// TIA Portal V17 export
// export: Created 2022-07-20T07:01:26.0319135Z, ExportSetting WithDefaults, DisplayName Totally Integrated Automation Portal, DisplayVersion V17, DisplayName TIA Portal Openness, DisplayVersion V17, DisplayName TIA Portal Version Control Interface, DisplayVersion V17, DisplayName SINAMICS Startdrive Advanced, DisplayVersion V17, DisplayName SINAMICS Startdrive G130, G150, S120, S150, SINAMICS MV, S210, DisplayVersion V17, DisplayName SINAMICS Startdrive G110M, G120, G120C, G120D, G120P, G115D, DisplayVersion V17, DisplayName STEP 7 Professional, DisplayVersion V17, DisplayName STEP 7 Safety, DisplayVersion V17, DisplayName WinCC Advanced, DisplayVersion V17
FUNCTION_BLOCK "FB10233_LAM_PositionningMotor"   // FB10233, LAD
{ S7_Optimized_Access := 'TRUE' }
VERSION : 0.1
// stored: AutoNumber false, IsIECCheckEnabled false, IsRetainMemResEnabled false, MemoryReserve 100, SetENOAutomatically false, UDAEnableTagReadback false
   VAR_INPUT
      DriveInLexium : "TLexium_MDrv_Drv2Plc";
      HomingSensor : Bool;
      MmByMotorTurn : LReal;
      HoldCurrent : SInt;
      RunCurrent : SInt;
      HomingSpeedMmBySec : Real;
      SpeedMmBySec : Real;
      AccelerationMmBySec2 : Real;
      DecelerationMmBySec2 : Real;
      JogSpeedMmBySec : Real;
      OriginPosition : Real;
      StandByPosition : Real;
      WorkingPosition : Real;
   END_VAR
   VAR_OUTPUT
      ActualPosition : Real;
      HomingInProgress : Bool;
      HomingDone : Bool;
      InOriginPosition : Bool;
      IsInStandByPosition : Bool;
      InWorkingPosition : Bool;
      MotorInError : Bool;
      ErrorCode : Array[0..9] of UInt;
   END_VAR
   VAR_IN_OUT
      DriveOutLexium : "TLexium_MDrv_Plc2Drv";
      RequestAcknowledge : Bool;
      RequestHoming : Bool;
      RequestGoToOriginPosition : Bool;
      RequestGoToStandByPosition : Bool;
      RequestGoToWorkingPosition : Bool;
      RequestStop : Bool;
   END_VAR
   VAR
      Motor_Struct : Struct
         In : Struct
            EnableMotor : Bool;
            MmByTurn : LReal;
            "HomingVelocity_mm.s-1" : Real;
            "Velocity_mm.s-1" : Real;
            "Acceleration_mm.s-2" : Real;
            "Deceleration_mm.s-2" : Real;
            "JogVelocity_mm.s-1" : Real;
            RequestHoming : Bool;
            RequestGoToPosition_1 : Bool;
            Position_1 : Real;
            RequestGoToPosition_2 : Bool;
            Position_2 : Real;
            RequestGoToPosition_3 : Bool;
            Position_3 : Real;
            RequestGoToPosition_4 : Bool;
            Position_4 : Real;
            RequestGoToPosition_5 : Bool;
            Position_5 : Real;
            RequestJogPositive : Bool;
            RequestJogNegative : Bool;
            Ack : Bool;
            RequestStop : Bool;
         END_STRUCT;
         Out : Struct
            ActualPosition_mm : Real;
            MotorEnabled : Bool;
            HomingInProgress : Bool;
            HomingDone : Bool;
            IsInPosition_1 : Bool;
            IsInPosition_2 : Bool;
            IsInPosition_3 : Bool;
            IsInPosition_4 : Bool;
            IsInPosition_5 : Bool;
            InError : Bool;
            ErrorCode : Array[0..9] of UInt;
         END_STRUCT;
      END_STRUCT;
      SendRequestAfterEnableOk : Bool;
      SendNewRequestOk : Bool;
      MotorMovementManagementStateDiagram : Int;
      R_TRIG_HomingSensor : R_TRIG;
      R_TRIG_RequestHoming : R_TRIG;
      R_TRIG_RequestGoToOriginPosition : R_TRIG;
      R_TRIG_RequestGoToRecoveryPosition { S7_SetPoint := 'True'} : R_TRIG;
      R_TRIG_RequestGoToWorkingPosition : R_TRIG;
      R_TRIG_HomingDone { S7_SetPoint := 'True'} : R_TRIG;
      TON_Motor_SendRequestAfterEnabled { S7_SetPoint := 'True'} : TON_TIME;
      TON_Motor_SendNewRequest { S7_SetPoint := 'True'} : TON_TIME;
      FB10234_LexiumMotor_Instance { S7_SetPoint := 'True'} : "FB10234_LexiumMotor";
   END_VAR
   VAR CONSTANT
      WAIT_FOR_MOTOR_MOVEMENT_REQUESTS : Int := 0;
      MOTOR_HOMING : Int := 10;
      MOTOR_GO_TO_ORIGIN_POSITION : Int := 20;
      MOTOR_GO_TO_RECOVERY_POSITION : Int := 30;
      MOTOR_GO_TO_WORKING_POSITION : Int := 40;
      MOTOR_MOVEMENT_REQUEST_DONE : Int := 50;
   END_VAR
BEGIN

REGION Network 1 (SCL): First Scan
   IF "FirstScan" THEN
       #Motor_Struct.In.EnableMotor := FALSE;
       #Motor_Struct.In.RequestHoming := FALSE;
       #Motor_Struct.In.RequestGoToPosition_1 := FALSE;
       #Motor_Struct.In.RequestGoToPosition_2 := FALSE;
       #HomingDone := FALSE;
       #InOriginPosition := FALSE;
       #InWorkingPosition := FALSE;
       #SendRequestAfterEnableOk := FALSE;
       #SendNewRequestOk := FALSE;
       #MotorMovementManagementStateDiagram := #WAIT_FOR_MOTOR_MOVEMENT_REQUESTS;
   END_IF;
END_REGION

REGION Network 2 (SCL): Edge Signals & Timers
   REGION EDGE SIGNALS
       #R_TRIG_HomingSensor(CLK := #HomingSensor);
       #R_TRIG_RequestHoming(CLK := #RequestHoming AND #MotorMovementManagementStateDiagram = #WAIT_FOR_MOTOR_MOVEMENT_REQUESTS);
       #R_TRIG_RequestGoToOriginPosition(CLK := #RequestGoToOriginPosition AND #MotorMovementManagementStateDiagram = #WAIT_FOR_MOTOR_MOVEMENT_REQUESTS);
       #R_TRIG_RequestGoToRecoveryPosition(CLK := #RequestGoToStandByPosition AND #MotorMovementManagementStateDiagram = #WAIT_FOR_MOTOR_MOVEMENT_REQUESTS);
       #R_TRIG_RequestGoToWorkingPosition(CLK := #RequestGoToWorkingPosition AND #MotorMovementManagementStateDiagram = #WAIT_FOR_MOTOR_MOVEMENT_REQUESTS);
       #R_TRIG_HomingDone(CLK := #Motor_Struct.Out.HomingDone);
   END_REGION

   REGION TIMERS
       #TON_Motor_SendRequestAfterEnabled(IN := #Motor_Struct.Out.MotorEnabled,
                                          PT := T#1s);
       #TON_Motor_SendNewRequest(IN := #MotorMovementManagementStateDiagram = #MOTOR_HOMING OR
                                 #MotorMovementManagementStateDiagram = #MOTOR_GO_TO_ORIGIN_POSITION OR
                                 #MotorMovementManagementStateDiagram = #MOTOR_GO_TO_WORKING_POSITION,
                                 PT := T#2s);

   END_REGION
END_REGION

REGION Network 3 (SCL): Cleaning Tray Commands Management
   //Motor Parameters Management
   #Motor_Struct.In.MmByTurn := #MmByMotorTurn;
   #Motor_Struct.In."HomingVelocity_mm.s-1" := #HomingSpeedMmBySec;
   #Motor_Struct.In."Velocity_mm.s-1" := #SpeedMmBySec;
   #Motor_Struct.In."Acceleration_mm.s-2" := #AccelerationMmBySec2;
   #Motor_Struct.In."Deceleration_mm.s-2" := #DecelerationMmBySec2;
   #Motor_Struct.In."JogVelocity_mm.s-1" := #JogSpeedMmBySec;

   //Motors Positions Management
   #Motor_Struct.In.Position_1 := #OriginPosition;
   #Motor_Struct.In.Position_2 := #WorkingPosition;
   #Motor_Struct.In.Position_3 := #StandByPosition;

   //Motor Acknowledge Management
   #Motor_Struct.In.Ack := #RequestAcknowledge;

   //Motor Request Management
   IF #TON_Motor_SendRequestAfterEnabled.Q THEN
       #SendRequestAfterEnableOk := TRUE;
   END_IF;
   IF #TON_Motor_SendNewRequest.Q THEN
       #SendNewRequestOk := TRUE;
   END_IF;
   #Motor_Struct.In.RequestStop := #RequestStop;
END_REGION

REGION Network 4: Motor Management
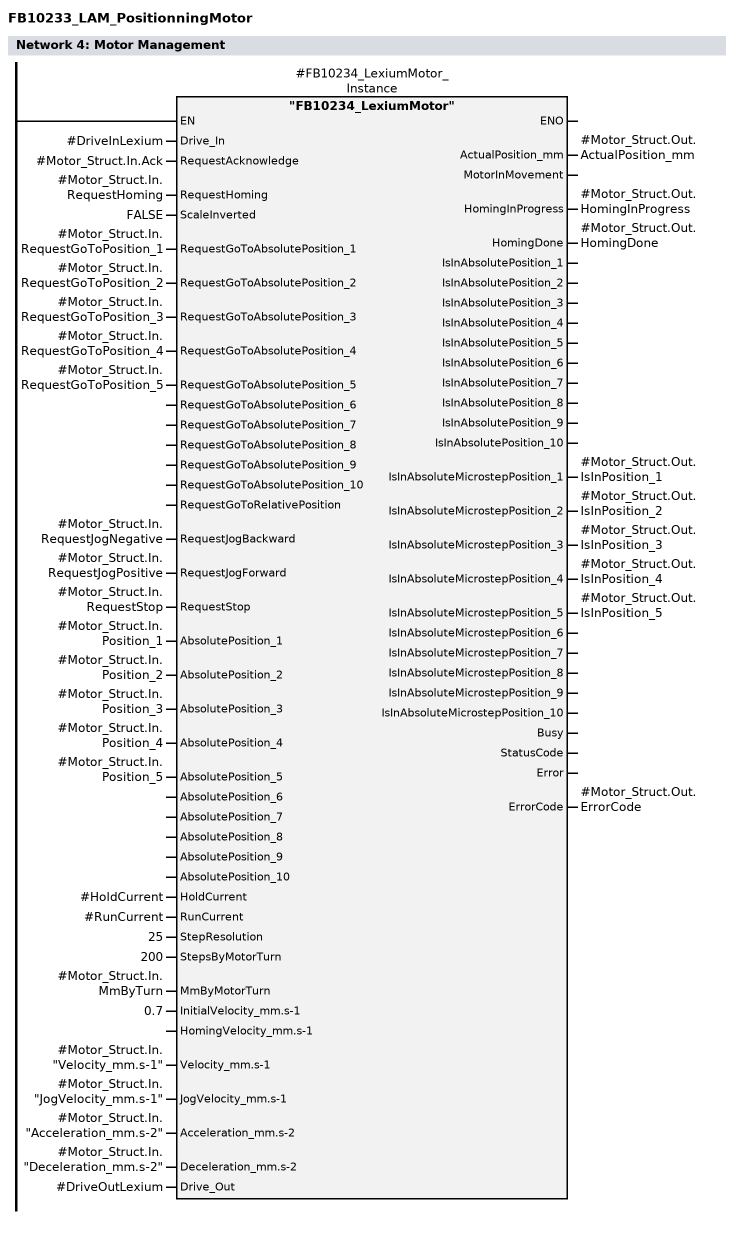
   RUNG wire#powerrail
      #FB10234_LexiumMotor_Instance(Drive_In := #DriveInLexium, RequestAcknowledge := #Motor_Struct.In.Ack, RequestHoming := #Motor_Struct.In.RequestHoming, ScaleInverted := FALSE, RequestGoToAbsolutePosition_1 := #Motor_Struct.In.RequestGoToPosition_1, RequestGoToAbsolutePosition_2 := #Motor_Struct.In.RequestGoToPosition_2, RequestGoToAbsolutePosition_3 := #Motor_Struct.In.RequestGoToPosition_3, RequestGoToAbsolutePosition_4 := #Motor_Struct.In.RequestGoToPosition_4, RequestGoToAbsolutePosition_5 := #Motor_Struct.In.RequestGoToPosition_5, RequestGoToAbsolutePosition_6 :=, RequestGoToAbsolutePosition_7 :=, RequestGoToAbsolutePosition_8 :=, RequestGoToAbsolutePosition_9 :=, RequestGoToAbsolutePosition_10 :=, RequestGoToRelativePosition :=, RequestJogBackward := #Motor_Struct.In.RequestJogNegative, RequestJogForward := #Motor_Struct.In.RequestJogPositive, RequestStop := #Motor_Struct.In.RequestStop, AbsolutePosition_1 := #Motor_Struct.In.Position_1, AbsolutePosition_2 := #Motor_Struct.In.Position_2, AbsolutePosition_3 := #Motor_Struct.In.Position_3, AbsolutePosition_4 := #Motor_Struct.In.Position_4, AbsolutePosition_5 := #Motor_Struct.In.Position_5, AbsolutePosition_6 :=, AbsolutePosition_7 :=, AbsolutePosition_8 :=, AbsolutePosition_9 :=, AbsolutePosition_10 :=, HoldCurrent := #HoldCurrent, RunCurrent := #RunCurrent, StepResolution := 25, StepsByMotorTurn := 200, MmByMotorTurn := #Motor_Struct.In.MmByTurn, "InitialVelocity_mm.s-1" := 0.7, "HomingVelocity_mm.s-1" :=, "Velocity_mm.s-1" := #Motor_Struct.In."Velocity_mm.s-1", "JogVelocity_mm.s-1" := #Motor_Struct.In."JogVelocity_mm.s-1", "Acceleration_mm.s-2" := #Motor_Struct.In."Acceleration_mm.s-2", "Deceleration_mm.s-2" := #Motor_Struct.In."Deceleration_mm.s-2", Drive_Out := #DriveOutLexium, ActualPosition_mm => #Motor_Struct.Out.ActualPosition_mm, MotorInMovement =>, HomingInProgress => #Motor_Struct.Out.HomingInProgress, HomingDone => #Motor_Struct.Out.HomingDone, IsInAbsolutePosition_1 =>, IsInAbsolutePosition_2 =>, IsInAbsolutePosition_3 =>, IsInAbsolutePosition_4 =>, IsInAbsolutePosition_5 =>, IsInAbsolutePosition_6 =>, IsInAbsolutePosition_7 =>, IsInAbsolutePosition_8 =>, IsInAbsolutePosition_9 =>, IsInAbsolutePosition_10 =>, IsInAbsoluteMicrostepPosition_1 => #Motor_Struct.Out.IsInPosition_1, IsInAbsoluteMicrostepPosition_2 => #Motor_Struct.Out.IsInPosition_2, IsInAbsoluteMicrostepPosition_3 => #Motor_Struct.Out.IsInPosition_3, IsInAbsoluteMicrostepPosition_4 => #Motor_Struct.Out.IsInPosition_4, IsInAbsoluteMicrostepPosition_5 => #Motor_Struct.Out.IsInPosition_5, IsInAbsoluteMicrostepPosition_6 =>, IsInAbsoluteMicrostepPosition_7 =>, IsInAbsoluteMicrostepPosition_8 =>, IsInAbsoluteMicrostepPosition_9 =>, IsInAbsoluteMicrostepPosition_10 =>, Busy =>, StatusCode =>, Error =>, ErrorCode => #Motor_Struct.Out.ErrorCode)
   END_RUNG
   // the same network as SCL:
   #FB10234_LexiumMotor_Instance(Drive_In := #DriveInLexium,   // "FB10234_LexiumMotor"
                           RequestAcknowledge := #Motor_Struct.In.Ack,
                           RequestHoming := #Motor_Struct.In.RequestHoming,
                           ScaleInverted := FALSE,
                           RequestGoToAbsolutePosition_1 := #Motor_Struct.In.RequestGoToPosition_1,
                           RequestGoToAbsolutePosition_2 := #Motor_Struct.In.RequestGoToPosition_2,
                           RequestGoToAbsolutePosition_3 := #Motor_Struct.In.RequestGoToPosition_3,
                           RequestGoToAbsolutePosition_4 := #Motor_Struct.In.RequestGoToPosition_4,
                           RequestGoToAbsolutePosition_5 := #Motor_Struct.In.RequestGoToPosition_5,
                           RequestJogBackward := #Motor_Struct.In.RequestJogNegative,
                           RequestJogForward := #Motor_Struct.In.RequestJogPositive,
                           RequestStop := #Motor_Struct.In.RequestStop,
                           AbsolutePosition_1 := #Motor_Struct.In.Position_1,
                           AbsolutePosition_2 := #Motor_Struct.In.Position_2,
                           AbsolutePosition_3 := #Motor_Struct.In.Position_3,
                           AbsolutePosition_4 := #Motor_Struct.In.Position_4,
                           AbsolutePosition_5 := #Motor_Struct.In.Position_5,
                           HoldCurrent := #HoldCurrent,
                           RunCurrent := #RunCurrent,
                           StepResolution := 25,
                           StepsByMotorTurn := 200,
                           MmByMotorTurn := #Motor_Struct.In.MmByTurn,
                           "InitialVelocity_mm.s-1" := 0.7,
                           "Velocity_mm.s-1" := #Motor_Struct.In."Velocity_mm.s-1",
                           "JogVelocity_mm.s-1" := #Motor_Struct.In."JogVelocity_mm.s-1",
                           "Acceleration_mm.s-2" := #Motor_Struct.In."Acceleration_mm.s-2",
                           "Deceleration_mm.s-2" := #Motor_Struct.In."Deceleration_mm.s-2",
                           Drive_Out := #DriveOutLexium,
                           ActualPosition_mm => #Motor_Struct.Out.ActualPosition_mm,
                           HomingInProgress => #Motor_Struct.Out.HomingInProgress,
                           HomingDone => #Motor_Struct.Out.HomingDone,
                           IsInAbsoluteMicrostepPosition_1 => #Motor_Struct.Out.IsInPosition_1,
                           IsInAbsoluteMicrostepPosition_2 => #Motor_Struct.Out.IsInPosition_2,
                           IsInAbsoluteMicrostepPosition_3 => #Motor_Struct.Out.IsInPosition_3,
                           IsInAbsoluteMicrostepPosition_4 => #Motor_Struct.Out.IsInPosition_4,
                           IsInAbsoluteMicrostepPosition_5 => #Motor_Struct.Out.IsInPosition_5,
                           ErrorCode => #Motor_Struct.Out.ErrorCode);
END_REGION

REGION Network 5 (SCL): Motor Movement Management
   IF #Motor_Struct.In.RequestStop THEN
       #MotorMovementManagementStateDiagram := #WAIT_FOR_MOTOR_MOVEMENT_REQUESTS;
       #Motor_Struct.In.RequestHoming := FALSE;
       #Motor_Struct.In.RequestJogPositive := FALSE;
       #Motor_Struct.In.RequestJogNegative := FALSE;
       #Motor_Struct.In.RequestGoToPosition_1 := FALSE;
       #Motor_Struct.In.RequestGoToPosition_2 := FALSE;
       #Motor_Struct.In.RequestGoToPosition_3 := FALSE;
       #Motor_Struct.In.RequestGoToPosition_4 := FALSE;
       #Motor_Struct.In.RequestGoToPosition_5 := FALSE;
   END_IF;

   CASE #MotorMovementManagementStateDiagram OF
       #WAIT_FOR_MOTOR_MOVEMENT_REQUESTS:
           IF #R_TRIG_RequestHoming.Q THEN
               #HomingDone := FALSE;
               #MotorMovementManagementStateDiagram := #MOTOR_HOMING;
           ELSIF #R_TRIG_RequestGoToOriginPosition.Q THEN
               #MotorMovementManagementStateDiagram := #MOTOR_GO_TO_ORIGIN_POSITION;
           ELSIF #R_TRIG_RequestGoToRecoveryPosition.Q THEN
               #MotorMovementManagementStateDiagram := #MOTOR_GO_TO_RECOVERY_POSITION;
           ELSIF #R_TRIG_RequestGoToWorkingPosition.Q THEN
               #MotorMovementManagementStateDiagram := #MOTOR_GO_TO_WORKING_POSITION;
           END_IF;
       #MOTOR_HOMING:
           #Motor_Struct.In.RequestHoming := TRUE;
           IF #R_TRIG_HomingDone.Q THEN
               #Motor_Struct.In.RequestHoming := FALSE;
               #SendNewRequestOk := FALSE;
               RESET_TIMER(#TON_Motor_SendNewRequest);
               #MotorMovementManagementStateDiagram := #MOTOR_MOVEMENT_REQUEST_DONE;
           END_IF;
       #MOTOR_GO_TO_ORIGIN_POSITION:
           #Motor_Struct.In.RequestGoToPosition_1 := TRUE;
           IF #Motor_Struct.Out.IsInPosition_1 THEN
               #Motor_Struct.In.RequestGoToPosition_1 := FALSE;
               RESET_TIMER(#TON_Motor_SendNewRequest);
               #MotorMovementManagementStateDiagram := #MOTOR_MOVEMENT_REQUEST_DONE;
           END_IF;
       #MOTOR_GO_TO_RECOVERY_POSITION:
           #Motor_Struct.In.RequestGoToPosition_3 := TRUE;
           IF #Motor_Struct.Out.IsInPosition_3 THEN
               #Motor_Struct.In.RequestGoToPosition_3 := FALSE;
               RESET_TIMER(#TON_Motor_SendNewRequest);
               #MotorMovementManagementStateDiagram := #MOTOR_MOVEMENT_REQUEST_DONE;
           END_IF;
       #MOTOR_GO_TO_WORKING_POSITION:
           #Motor_Struct.In.RequestGoToPosition_2 := TRUE;
           IF #Motor_Struct.Out.IsInPosition_2 THEN
               #Motor_Struct.In.RequestGoToPosition_2 := FALSE;
               RESET_TIMER(#TON_Motor_SendNewRequest);
               #MotorMovementManagementStateDiagram := #MOTOR_MOVEMENT_REQUEST_DONE;
           END_IF;

       #MOTOR_MOVEMENT_REQUEST_DONE:
           #MotorMovementManagementStateDiagram := #WAIT_FOR_MOTOR_MOVEMENT_REQUESTS;
   END_CASE;
END_REGION

REGION Network 6 (SCL): Motor Error Management
   IF #Motor_Struct.Out.InError THEN
       #MotorMovementManagementStateDiagram := #WAIT_FOR_MOTOR_MOVEMENT_REQUESTS;
       #Motor_Struct.In.Ack := #RequestAcknowledge;
       #Motor_Struct.In.EnableMotor := FALSE;
       #Motor_Struct.In.RequestHoming := FALSE;
       #Motor_Struct.In.RequestGoToPosition_1 := FALSE;
       #Motor_Struct.In.RequestGoToPosition_2 := FALSE;
       #SendRequestAfterEnableOk := FALSE;
       #SendNewRequestOk := FALSE;
       #HomingDone := FALSE;
   END_IF;
END_REGION

REGION Network 7 (SCL): Trays States Management
   //Motor Position States Management
   #ActualPosition := #Motor_Struct.Out.ActualPosition_mm;
   #InOriginPosition := #Motor_Struct.Out.IsInPosition_1;
   #InWorkingPosition := #Motor_Struct.Out.IsInPosition_2;
   #IsInStandByPosition := #Motor_Struct.Out.IsInPosition_3;

   //Motor Error States Management
   #HomingInProgress := #Motor_Struct.Out.HomingInProgress;
   #HomingDone := #Motor_Struct.Out.HomingDone;
   #MotorInError := #Motor_Struct.Out.InError;
   #ErrorCode := #Motor_Struct.Out.ErrorCode;
END_REGION
END_FUNCTION_BLOCK
